FUNCTION SPLIT_LWORD_INTO_BOOLS (* this Function extracts the 64 BOOLS from a lword *)
  (* Standard: 61499-1; Description: Copyright (c) 2024 HR Agrartechnik GmbH This program and the accompanying materials are made available under the terms of the Eclipse Public License 2.0 which is available at https://www.eclipse.org/legal/epl-2.0/ SPDX-License-Identifier: EPL-2.0 *)
  (* Version 1.0, 2024-02-22, Franz Höpfinger, HR Agrartechnik, initial Implementation *)
  (* Version 1.1, 2024-07-24, Moritz Ortmeier, HR Agrartechnik, rename Function and change Output Variables *)
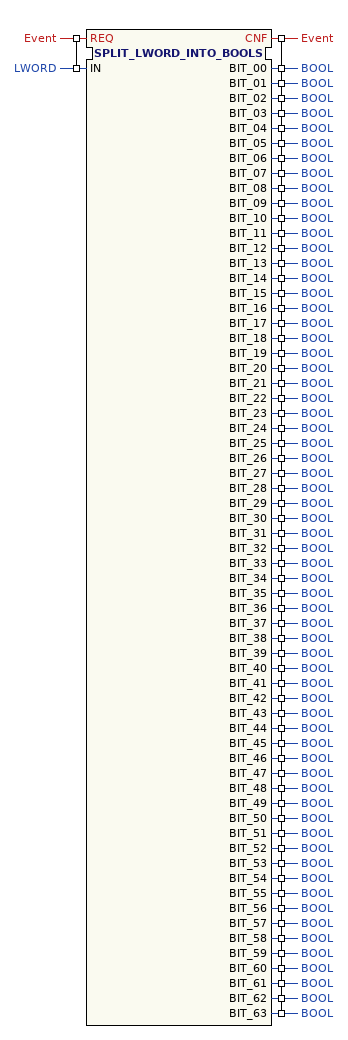
  EVENT_INPUT
    REQ WITH IN; (* Normal Execution Request *)
  END_EVENT
  EVENT_OUTPUT
    CNF WITH BIT_00, BIT_01, BIT_02, BIT_03, BIT_04, BIT_05, BIT_06, BIT_07, BIT_08, BIT_09, BIT_10, BIT_11, BIT_12, BIT_13, BIT_14, BIT_15, BIT_16, BIT_17, BIT_18, BIT_19, BIT_20, BIT_21, BIT_22, BIT_23, BIT_24, BIT_25, BIT_26, BIT_27, BIT_28, BIT_29, BIT_30, BIT_31, BIT_32, BIT_33, BIT_34, BIT_35, BIT_36, BIT_37, BIT_38, BIT_39, BIT_40, BIT_41, BIT_42, BIT_43, BIT_44, BIT_45, BIT_46, BIT_47, BIT_48, BIT_49, BIT_50, BIT_51, BIT_52, BIT_53, BIT_54, BIT_55, BIT_56, BIT_57, BIT_58, BIT_59, BIT_60, BIT_61, BIT_62, BIT_63; (* Execution Confirmation *)
  END_EVENT
  VAR_INPUT
    IN : LWORD;
  END_VAR
  VAR_OUTPUT
    BIT_00 : BOOL;
    BIT_01 : BOOL;
    BIT_02 : BOOL;
    BIT_03 : BOOL;
    BIT_04 : BOOL;
    BIT_05 : BOOL;
    BIT_06 : BOOL;
    BIT_07 : BOOL;
    BIT_08 : BOOL;
    BIT_09 : BOOL;
    BIT_10 : BOOL;
    BIT_11 : BOOL;
    BIT_12 : BOOL;
    BIT_13 : BOOL;
    BIT_14 : BOOL;
    BIT_15 : BOOL;
    BIT_16 : BOOL;
    BIT_17 : BOOL;
    BIT_18 : BOOL;
    BIT_19 : BOOL;
    BIT_20 : BOOL;
    BIT_21 : BOOL;
    BIT_22 : BOOL;
    BIT_23 : BOOL;
    BIT_24 : BOOL;
    BIT_25 : BOOL;
    BIT_26 : BOOL;
    BIT_27 : BOOL;
    BIT_28 : BOOL;
    BIT_29 : BOOL;
    BIT_30 : BOOL;
    BIT_31 : BOOL;
    BIT_32 : BOOL;
    BIT_33 : BOOL;
    BIT_34 : BOOL;
    BIT_35 : BOOL;
    BIT_36 : BOOL;
    BIT_37 : BOOL;
    BIT_38 : BOOL;
    BIT_39 : BOOL;
    BIT_40 : BOOL;
    BIT_41 : BOOL;
    BIT_42 : BOOL;
    BIT_43 : BOOL;
    BIT_44 : BOOL;
    BIT_45 : BOOL;
    BIT_46 : BOOL;
    BIT_47 : BOOL;
    BIT_48 : BOOL;
    BIT_49 : BOOL;
    BIT_50 : BOOL;
    BIT_51 : BOOL;
    BIT_52 : BOOL;
    BIT_53 : BOOL;
    BIT_54 : BOOL;
    BIT_55 : BOOL;
    BIT_56 : BOOL;
    BIT_57 : BOOL;
    BIT_58 : BOOL;
    BIT_59 : BOOL;
    BIT_60 : BOOL;
    BIT_61 : BOOL;
    BIT_62 : BOOL;
    BIT_63 : BOOL;
  END_VAR
  BODY IN ST:
(* this Function extracts the 64 BOOLS from a lword *)
FUNCTION SPLIT_LWORD_INTO_BOOLS

VAR_INPUT
	IN : LWORD;
END_VAR

VAR_OUTPUT
	BIT_00 : BOOL;
	BIT_01 : BOOL;
	BIT_02 : BOOL;
	BIT_03 : BOOL;
	BIT_04 : BOOL;
	BIT_05 : BOOL;
	BIT_06 : BOOL;
	BIT_07 : BOOL;
	BIT_08 : BOOL;
	BIT_09 : BOOL;
	BIT_10 : BOOL;
	BIT_11 : BOOL;
	BIT_12 : BOOL;
	BIT_13 : BOOL;
	BIT_14 : BOOL;
	BIT_15 : BOOL;
	BIT_16 : BOOL;
	BIT_17 : BOOL;
	BIT_18 : BOOL;
	BIT_19 : BOOL;
	BIT_20 : BOOL;
	BIT_21 : BOOL;
	BIT_22 : BOOL;
	BIT_23 : BOOL;
	BIT_24 : BOOL;
	BIT_25 : BOOL;
	BIT_26 : BOOL;
	BIT_27 : BOOL;
	BIT_28 : BOOL;
	BIT_29 : BOOL;
	BIT_30 : BOOL;
	BIT_31 : BOOL;
	BIT_32 : BOOL;
	BIT_33 : BOOL;
	BIT_34 : BOOL;
	BIT_35 : BOOL;
	BIT_36 : BOOL;
	BIT_37 : BOOL;
	BIT_38 : BOOL;
	BIT_39 : BOOL;
	BIT_40 : BOOL;
	BIT_41 : BOOL;
	BIT_42 : BOOL;
	BIT_43 : BOOL;
	BIT_44 : BOOL;
	BIT_45 : BOOL;
	BIT_46 : BOOL;
	BIT_47 : BOOL;
	BIT_48 : BOOL;
	BIT_49 : BOOL;
	BIT_50 : BOOL;
	BIT_51 : BOOL;
	BIT_52 : BOOL;
	BIT_53 : BOOL;
	BIT_54 : BOOL;
	BIT_55 : BOOL;
	BIT_56 : BOOL;
	BIT_57 : BOOL;
	BIT_58 : BOOL;
	BIT_59 : BOOL;
	BIT_60 : BOOL;
	BIT_61 : BOOL;
	BIT_62 : BOOL;
	BIT_63 : BOOL;
END_VAR

BIT_00 := IN.%X0;
BIT_01 := IN.%X1;
BIT_02 := IN.%X2;
BIT_03 := IN.%X3;
BIT_04 := IN.%X4;
BIT_05 := IN.%X5;
BIT_06 := IN.%X6;
BIT_07 := IN.%X7;
BIT_08 := IN.%X8;
BIT_09 := IN.%X9;
BIT_10 := IN.%X10;
BIT_11 := IN.%X11;
BIT_12 := IN.%X12;
BIT_13 := IN.%X13;
BIT_14 := IN.%X14;
BIT_15 := IN.%X15;
BIT_16 := IN.%X16;
BIT_17 := IN.%X17;
BIT_18 := IN.%X18;
BIT_19 := IN.%X19;
BIT_20 := IN.%X20;
BIT_21 := IN.%X21;
BIT_22 := IN.%X22;
BIT_23 := IN.%X23;
BIT_24 := IN.%X24;
BIT_25 := IN.%X25;
BIT_26 := IN.%X26;
BIT_27 := IN.%X27;
BIT_28 := IN.%X28;
BIT_29 := IN.%X29;
BIT_30 := IN.%X30;
BIT_31 := IN.%X31;
BIT_32 := IN.%X32;
BIT_33 := IN.%X33;
BIT_34 := IN.%X34;
BIT_35 := IN.%X35;
BIT_36 := IN.%X36;
BIT_37 := IN.%X37;
BIT_38 := IN.%X38;
BIT_39 := IN.%X39;
BIT_40 := IN.%X40;
BIT_41 := IN.%X41;
BIT_42 := IN.%X42;
BIT_43 := IN.%X43;
BIT_44 := IN.%X44;
BIT_45 := IN.%X45;
BIT_46 := IN.%X46;
BIT_47 := IN.%X47;
BIT_48 := IN.%X48;
BIT_49 := IN.%X49;
BIT_50 := IN.%X50;
BIT_51 := IN.%X51;
BIT_52 := IN.%X52;
BIT_53 := IN.%X53;
BIT_54 := IN.%X54;
BIT_55 := IN.%X55;
BIT_56 := IN.%X56;
BIT_57 := IN.%X57;
BIT_58 := IN.%X58;
BIT_59 := IN.%X59;
BIT_60 := IN.%X60;
BIT_61 := IN.%X61;
BIT_62 := IN.%X62;
BIT_63 := IN.%X63;
END_FUNCTION
  END_BODY
END_FUNCTION
